// TIA Portal project "2020-10-09_TestRilevatoreFronte" (V16)

(* hardware
DEVICE "S7-1200 station_1"  S7-1200 Station
   slot 0: "Telaio di montaggio_0"  S7-1200 Rack  Rack  V1.0
   slot 1: "PLC_1"  CPU 1215C DC/DC/DC  6ES7 215-1AG40-0XB0  V4.4
*)

// ===== PLC "PLC_1"  CPU 1215C DC/DC/DC =====

VAR_GLOBAL   // PLC tag table "Tabella delle variabili standard"
   "lampada" AT %Q0.0 : Bool;
   "sirenaFineTurno" AT %Q0.1 : Bool;
   "segnaleFineTurno" AT %I0.2 : Bool;
   "spegni" AT %I0.1 : Bool;
   "accendi" AT %I0.0 : Bool;
   "spegni_old" AT %M0.0 : Bool;
   "segnaleFineTurno_old" AT %M0.1 : Bool;
   "segnaleFineTurno_old2" AT %M0.2 : Bool;
END_VAR

ORGANIZATION_BLOCK "Main"   // OB1, LAD, ProgramCycle
TITLE = "Main Program Sweep (Cycle)"
{ S7_Optimized_Access := 'TRUE' }
VERSION : 0.1
   VAR_INPUT
      Initial_Call : Bool;   // Initial call of this OB
      Remanence : Bool;   // =True, if remanent data are available
   END_VAR
   VAR_TEMP   // added for the SCL form of the ladder/FBD networks
      _w1 : Bool;
      _w2 : Bool;
   END_VAR
BEGIN

REGION Network 1: spegnimento lampada con interblocco
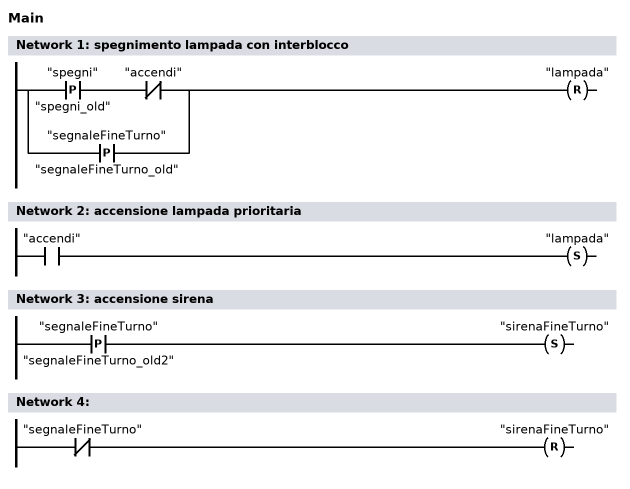
   RUNG wire#powerrail
      P_Contact(operand := "spegni", bit := "spegni_old")
      I_Contact( "accendi" )
      wire#w1
      R_Coil( "lampada" )
   END_RUNG
   RUNG wire#powerrail
      P_Contact(operand := "segnaleFineTurno", bit := "segnaleFineTurno_old")
   END_RUNG wire#w1
   // the same network as SCL:
   #_w1 := "spegni" AND NOT "spegni_old";   // rising edge of "spegni"
   "spegni_old" := "spegni";
   #_w2 := "segnaleFineTurno" AND NOT "segnaleFineTurno_old";   // rising edge of "segnaleFineTurno"
   "segnaleFineTurno_old" := "segnaleFineTurno";
   IF (#_w1 AND NOT "accendi") OR #_w2 THEN "lampada" := FALSE; END_IF;
END_REGION

REGION Network 2: accensione lampada prioritaria
   RUNG wire#powerrail
      Contact( "accendi" )
      S_Coil( "lampada" )
   END_RUNG
   // the same network as SCL:
   IF "accendi" THEN "lampada" := TRUE; END_IF;
END_REGION

REGION Network 3: accensione sirena
   RUNG wire#powerrail
      P_Contact(operand := "segnaleFineTurno", bit := "segnaleFineTurno_old2")
      S_Coil( "sirenaFineTurno" )
   END_RUNG
   // the same network as SCL:
   #_w1 := "segnaleFineTurno" AND NOT "segnaleFineTurno_old2";   // rising edge of "segnaleFineTurno"
   "segnaleFineTurno_old2" := "segnaleFineTurno";
   IF #_w1 THEN "sirenaFineTurno" := TRUE; END_IF;
END_REGION

REGION Network 4
   RUNG wire#powerrail
      I_Contact( "segnaleFineTurno" )
      R_Coil( "sirenaFineTurno" )
   END_RUNG
   // the same network as SCL:
   IF NOT "segnaleFineTurno" THEN "sirenaFineTurno" := FALSE; END_IF;
END_REGION
END_ORGANIZATION_BLOCK